Yaskawa INFORM job: DEMO_ROOF_SIDE_0625_3.JBI

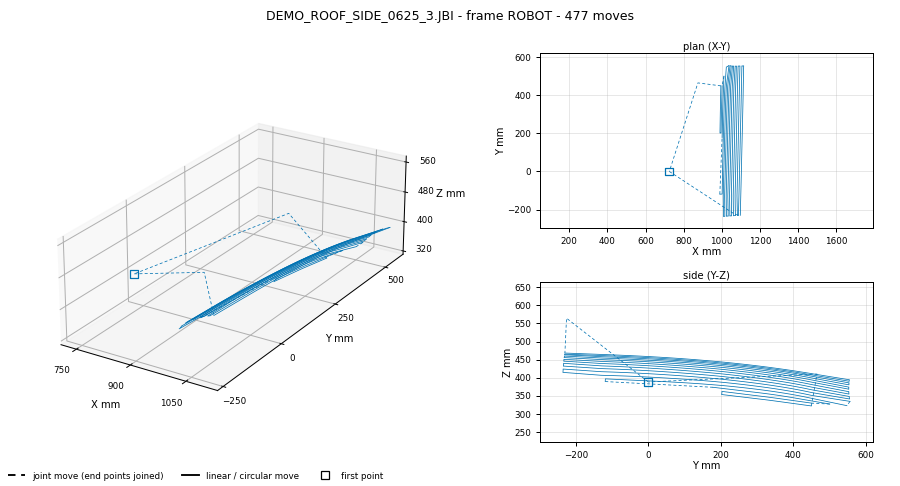
[picture p0: tool path of DEMO_ROOF_SIDE_0625_3.JBI in frame ROBOT, 477 of 477 moves have a stored position in this frame; points joined in program order, loops and branches not executed]
/JOB
//NAME DEMO_ROOF_SIDE_0625_3
//POS
///NPOS 477,0,0,0,0,0
///TOOL 0
///USER 0
///POSTYPE ROBOT
///RECTAN
///RCONF 1,0,0,0,0,0,0,0,0,0,0,0,0,0,0,0,0,0,0,0,0,0,0,0
C00000=725.000,0.000,388.500,-180.000,-0.000,0.000
///USER 0
///POSTYPE ROBOT
///RECTAN
C00001=1070.165,-225.804,564.348,177.658,-15.895,-0.730
C00002=1097.475,-230.239,468.252,177.658,-15.895,-0.730
C00003=1100.518,-106.522,463.583,177.658,-15.895,-0.730
C00004=1101.131,-81.381,462.555,177.457,-15.868,-0.652
C00005=1101.733,-56.230,461.444,177.242,-15.858,-0.568
C00006=1102.322,-31.102,460.246,177.018,-15.859,-0.492
C00007=1102.894,-6.471,458.979,176.786,-15.861,-0.417
C00008=1103.450,17.667,457.639,176.549,-15.857,-0.346
C00009=1103.994,41.321,456.228,176.307,-15.841,-0.282
C00010=1104.527,64.471,454.750,176.060,-15.805,-0.220
C00011=1105.052,87.116,453.204,175.808,-15.748,-0.164
C00012=1105.569,109.258,451.595,175.550,-15.665,-0.106
C00013=1106.076,130.831,449.928,175.291,-15.558,-0.055
C00014=1106.579,151.961,448.197,175.027,-15.428,-0.007
C00015=1107.074,172.585,446.411,174.761,-15.276,0.037
C00016=1107.562,192.652,444.578,174.493,-15.108,0.083
C00017=1107.979,209.697,442.942,174.219,-14.948,0.167
C00018=1108.302,223.398,441.579,174.012,-14.865,0.226
C00019=1108.743,242.055,439.641,173.727,-14.761,0.293
C00020=1109.169,260.166,437.673,173.443,-14.671,0.359
C00021=1109.576,277.536,435.703,173.164,-14.597,0.432
C00022=1109.980,294.921,433.649,172.877,-14.541,0.511
C00023=1110.375,312.126,431.533,172.586,-14.508,0.594
C00024=1110.754,328.858,429.397,172.296,-14.503,0.687
C00025=1111.108,344.779,427.292,172.012,-14.528,0.783
C00026=1111.443,360.182,425.185,171.727,-14.588,0.893
C00027=1111.759,375.112,423.077,171.442,-14.686,1.009
C00028=1112.046,389.128,421.040,171.165,-14.822,1.140
C00029=1112.303,402.245,419.083,170.893,-14.997,1.282
C00030=1112.529,414.390,417.227,170.620,-15.203,1.466
C00031=1112.829,431.883,414.478,170.211,-15.618,1.704
C00032=1112.994,442.551,412.752,169.934,-15.944,1.913
C00033=1113.129,452.452,411.121,169.867,-16.412,1.571
C00034=1115.209,553.765,394.636,169.867,-16.412,1.571
C00035=1105.880,553.291,390.560,169.867,-16.412,1.571
C00036=1103.548,452.102,407.760,170.054,-16.524,0.911
C00037=1103.388,442.223,409.459,170.213,-16.114,0.900
C00038=1103.203,431.578,411.246,170.442,-15.758,0.852
C00039=1103.095,425.743,412.205,170.567,-15.593,0.818
C00040=1102.875,414.111,414.077,170.805,-15.314,0.762
C00041=1102.635,401.997,415.975,171.043,-15.085,0.705
C00042=1102.366,388.898,417.968,171.291,-14.896,0.647
C00043=1102.069,374.899,420.034,171.548,-14.747,0.593
C00044=1101.745,359.987,422.164,171.815,-14.637,0.542
C00045=1101.405,344.600,424.286,172.084,-14.567,0.497
C00046=1101.047,328.694,426.405,172.354,-14.533,0.455
C00047=1100.666,311.978,428.548,172.631,-14.531,0.417
C00048=1100.269,294.786,430.667,172.910,-14.557,0.381
C00049=1099.865,277.416,432.721,173.185,-14.607,0.348
C00050=1099.459,260.059,434.689,173.454,-14.675,0.317
C00051=1099.033,241.963,436.653,173.728,-14.762,0.287
C00052=1098.594,223.318,438.585,174.004,-14.862,0.256
C00053=1098.272,209.617,439.948,174.202,-14.941,0.233
C00054=1097.859,192.596,441.565,174.459,-15.096,0.211
C00055=1097.377,172.542,443.383,174.722,-15.263,0.186
C00056=1096.886,151.931,445.156,174.983,-15.414,0.158
C00057=1096.387,130.814,446.876,175.242,-15.544,0.128
C00058=1095.880,109.241,448.536,175.496,-15.650,0.094
C00059=1095.365,87.114,450.143,175.748,-15.732,0.058
C00060=1094.841,64.483,451.688,175.995,-15.790,0.019
C00061=1094.306,41.347,453.169,176.236,-15.824,-0.022
C00062=1093.761,17.708,454.585,176.472,-15.841,-0.065
C00063=1093.202,-6.416,455.932,176.701,-15.844,-0.107
C00064=1092.628,-31.032,457.209,176.924,-15.841,-0.148
C00065=1092.035,-56.147,458.416,177.138,-15.840,-0.185
C00066=1091.433,-81.271,459.530,177.338,-15.849,-0.214
C00067=1090.821,-106.401,460.556,177.519,-15.875,-0.223
C00068=1087.825,-230.592,465.270,177.627,-15.905,-0.084
C00069=1082.226,-231.045,463.513,177.619,-15.904,-0.053
C00070=1080.117,-128.026,458.207,177.788,-18.751,-0.644
C00071=1080.712,-103.412,457.271,177.590,-18.756,-0.572
C00072=1081.269,-80.191,456.312,177.387,-18.785,-0.479
C00073=1081.838,-56.094,455.234,177.168,-18.840,-0.381
C00074=1082.398,-31.914,454.063,176.940,-18.915,-0.284
C00075=1082.945,-7.981,452.812,176.706,-19.000,-0.187
C00076=1083.496,16.375,451.444,176.461,-19.092,-0.091
C00077=1084.037,40.477,449.991,176.212,-19.178,-0.000
C00078=1084.553,63.576,448.505,175.965,-19.251,0.090
C00079=1085.072,86.781,446.916,175.707,-19.310,0.180
C00080=1085.565,108.870,445.310,175.452,-19.348,0.267
C00081=1086.061,131.068,443.602,175.187,-19.367,0.355
C00082=1086.534,152.148,441.887,174.923,-19.366,0.439
C00083=1087.008,173.221,440.078,174.650,-19.349,0.524
C00084=1087.464,193.399,438.254,174.377,-19.320,0.605
C00085=1087.825,209.395,436.742,174.074,-19.286,0.725
C00086=1088.182,225.416,435.143,173.821,-19.308,0.819
C00087=1088.592,243.865,433.219,173.522,-19.338,0.924
C00088=1089.002,262.278,431.205,173.214,-19.372,1.033
C00089=1089.399,280.152,429.159,172.905,-19.415,1.143
C00090=1089.786,297.588,427.075,172.594,-19.469,1.257
C00091=1090.152,314.076,425.019,172.286,-19.535,1.380
C00092=1090.514,330.569,422.878,171.969,-19.624,1.504
C00093=1090.865,346.565,420.717,171.645,-19.736,1.643
C00094=1091.178,361.013,418.691,171.337,-19.865,1.785
C00095=1091.488,375.512,416.582,171.014,-20.031,1.934
C00096=1091.776,389.121,414.533,170.690,-20.226,2.100
C00097=1092.039,401.783,412.560,170.369,-20.450,2.275
C00098=1092.276,413.455,410.683,170.051,-20.704,2.449
C00099=1092.473,423.358,409.042,169.750,-20.957,2.640
C00100=1092.681,434.084,407.209,169.402,-21.286,2.853
C00101=1092.850,443.075,405.627,169.082,-21.612,3.061
C00102=1093.012,451.962,404.020,169.028,-22.108,2.662
C00103=1095.618,553.013,386.060,169.028,-22.108,2.662
C00104=1085.968,552.705,380.579,169.028,-22.108,2.662
C00105=1082.961,451.807,399.317,168.467,-27.285,2.821
C00106=1082.764,442.923,401.001,168.744,-26.842,2.800
C00107=1082.571,434.067,402.629,169.055,-26.469,2.748
C00108=1082.357,424.236,404.377,169.383,-26.117,2.669
C00109=1082.140,414.335,406.080,169.691,-25.812,2.584
C00110=1081.885,402.576,408.036,170.028,-25.504,2.481
C00111=1081.627,390.820,409.924,170.342,-25.243,2.382
C00112=1081.349,378.124,411.892,170.659,-25.004,2.281
C00113=1081.051,364.541,413.925,170.977,-24.787,2.181
C00114=1080.732,350.019,416.018,171.299,-24.590,2.080
C00115=1080.392,334.507,418.168,171.624,-24.411,1.978
C00116=1080.051,318.965,420.239,171.932,-24.254,1.881
C00117=1079.696,302.745,422.315,172.240,-24.111,1.786
C00118=1079.335,286.239,424.342,172.541,-23.978,1.692
C00119=1078.955,268.767,426.399,172.846,-23.847,1.597
C00120=1078.574,251.297,428.367,173.141,-23.722,1.504
C00121=1078.184,233.235,430.313,173.435,-23.593,1.410
C00122=1077.972,223.469,431.328,173.591,-23.524,1.360
C00123=1077.662,209.105,432.776,173.813,-23.421,1.287
C00124=1077.268,190.976,434.497,174.164,-23.354,1.206
C00125=1076.809,169.900,436.402,174.444,-23.276,1.116
C00126=1076.348,148.818,438.211,174.710,-23.191,1.028
C00127=1075.863,126.605,440.020,174.978,-23.092,0.939
C00128=1075.381,104.512,441.722,175.235,-22.981,0.852
C00129=1074.873,81.414,443.402,175.491,-22.854,0.763
C00130=1074.360,58.187,444.995,175.741,-22.715,0.676
C00131=1073.847,35.079,446.485,175.981,-22.572,0.593
C00132=1073.327,11.848,447.891,176.217,-22.427,0.511
C00133=1072.805,-11.255,449.199,176.446,-22.288,0.435
C00134=1072.275,-34.458,450.423,176.669,-22.160,0.365
C00135=1071.739,-57.560,451.554,176.884,-22.052,0.305
C00136=1071.195,-80.670,452.601,177.089,-21.967,0.257
C00137=1070.662,-102.916,453.529,177.273,-21.914,0.231
C00138=1070.057,-128.042,454.489,177.461,-21.888,0.238
C00139=1071.695,-231.567,459.915,177.355,-21.861,0.543
C00140=1061.501,-232.092,455.769,177.350,-21.861,0.556
C00141=1060.147,-128.074,450.149,177.673,-25.493,-0.352
C00142=1060.424,-116.502,449.716,177.561,-25.496,-0.306
C00143=1060.951,-94.862,448.854,177.335,-25.521,-0.191
C00144=1061.460,-73.669,447.935,177.106,-25.578,-0.067
C00145=1061.974,-51.990,446.914,176.870,-25.664,0.054
C00146=1062.492,-29.881,445.792,176.628,-25.776,0.181
C00147=1063.006,-7.714,444.584,176.382,-25.909,0.311
C00148=1063.527,14.959,443.259,176.128,-26.061,0.445
C00149=1064.053,38.144,441.813,175.866,-26.225,0.588
C00150=1064.574,61.324,440.273,175.600,-26.394,0.727
C00151=1065.091,84.498,438.639,175.330,-26.562,0.869
C00152=1065.593,107.167,436.947,175.056,-26.723,1.016
C00153=1066.079,129.265,435.203,174.777,-26.874,1.165
C00154=1066.552,150.925,433.402,174.490,-27.018,1.316
C00155=1067.011,172.078,431.549,174.196,-27.155,1.468
C00156=1067.457,192.659,429.652,173.895,-27.288,1.615
C00157=1067.805,208.750,428.099,173.466,-27.386,1.843
C00158=1068.310,232.062,425.676,173.073,-27.623,2.036
C00159=1068.730,251.306,423.568,172.729,-27.809,2.207
C00160=1069.116,268.867,421.555,172.398,-27.974,2.377
C00161=1069.505,286.433,419.452,172.047,-28.138,2.558
C00162=1069.874,303.035,417.377,171.699,-28.297,2.739
C00163=1070.242,319.454,415.238,171.336,-28.464,2.927
C00164=1070.595,335.095,413.114,170.965,-28.634,3.123
C00165=1070.927,349.716,411.048,170.598,-28.812,3.311
C00166=1071.240,363.349,409.047,170.224,-28.996,3.517
C00167=1071.559,377.040,406.959,169.821,-29.207,3.734
C00168=1071.859,389.849,404.929,169.410,-29.434,3.960
C00169=1072.142,401.720,402.976,168.993,-29.677,4.190
C00170=1072.406,412.613,401.117,168.564,-29.930,4.439
C00171=1072.674,423.498,399.190,168.090,-30.222,4.706
C00172=1072.925,433.455,397.359,167.603,-30.529,4.984
C00173=1073.167,442.803,395.573,167.144,-30.880,5.170
C00174=1073.417,451.686,393.819,167.000,-31.383,4.760
C00175=1076.941,552.431,374.355,167.000,-31.383,4.760
C00176=1070.604,552.364,368.674,167.000,-31.383,4.760
C00177=1064.303,450.677,387.868,166.732,-35.182,4.427
C00178=1063.991,441.090,389.826,167.182,-34.765,4.439
C00179=1063.720,432.199,391.572,167.581,-34.434,4.400
C00180=1063.453,423.074,393.298,167.968,-34.139,4.326
C00181=1063.171,413.034,395.127,168.363,-33.856,4.229
C00182=1062.875,402.145,397.038,168.761,-33.591,4.109
C00183=1062.585,391.123,398.901,169.134,-33.357,3.985
C00184=1062.277,379.170,400.848,169.505,-33.134,3.857
C00185=1061.955,366.340,402.861,169.871,-32.924,3.727
C00186=1061.623,352.844,404.897,170.232,-32.729,3.590
C00187=1061.284,338.827,406.933,170.580,-32.548,3.454
C00188=1060.933,324.057,408.996,170.921,-32.374,3.318
C00189=1060.562,308.264,411.115,171.264,-32.203,3.179
C00190=1060.195,292.480,413.150,171.585,-32.039,3.045
C00191=1059.791,274.985,415.313,171.923,-31.862,2.901
C00192=1059.578,265.654,416.429,172.096,-31.768,2.826
C00193=1059.153,246.982,418.589,172.428,-31.577,2.677
C00194=1058.723,227.872,420.701,172.753,-31.373,2.528
C00195=1058.283,208.328,422.764,173.071,-31.153,2.375
C00196=1057.996,195.285,424.047,173.443,-31.051,2.282
C00197=1057.574,176.199,425.849,173.723,-30.911,2.154
C00198=1057.126,155.969,427.670,174.001,-30.768,2.025
C00199=1056.654,134.875,429.477,174.275,-30.621,1.897
C00200=1056.157,112.776,431.275,174.547,-30.468,1.768
C00201=1055.652,90.530,432.991,174.809,-30.313,1.642
C00202=1055.123,67.421,434.676,175.073,-30.153,1.517
C00203=1054.608,45.164,436.208,175.322,-30.002,1.402
C00204=1054.092,23.041,437.644,175.565,-29.858,1.293
C00205=1053.572,0.919,438.994,175.807,-29.724,1.189
C00206=1053.043,-21.324,440.263,176.047,-29.606,1.091
C00207=1052.537,-42.438,441.385,176.272,-29.511,1.008
C00208=1052.052,-62.559,442.379,176.482,-29.443,0.939
C00209=1051.536,-83.822,443.351,176.696,-29.396,0.884
C00210=1051.017,-104.972,444.237,176.893,-29.379,0.856
C00211=1050.452,-128.121,445.120,177.078,-29.394,0.882
C00212=1051.564,-232.631,450.944,176.858,-29.343,1.365
C00213=1042.728,-233.148,445.881,176.855,-29.343,1.373
C00214=1041.055,-129.188,439.415,176.733,-33.542,1.452
C00215=1041.065,-127.686,439.343,177.520,-33.611,0.006
C00216=1041.589,-106.531,438.551,177.251,-33.551,0.150
C00217=1042.089,-86.375,437.718,176.986,-33.524,0.299
C00218=1042.591,-66.101,436.801,176.722,-33.523,0.444
C00219=1043.089,-45.974,435.813,176.456,-33.546,0.600
C00220=1043.609,-24.854,434.695,176.181,-33.593,0.760
C00221=1044.128,-3.735,433.493,175.906,-33.658,0.928
C00222=1044.670,18.526,432.137,175.625,-33.744,1.095
C00223=1045.207,40.652,430.701,175.342,-33.840,1.273
C00224=1045.742,62.918,429.165,175.060,-33.945,1.448
C00225=1046.270,85.031,427.551,174.774,-34.054,1.631
C00226=1046.792,107.138,425.848,174.479,-34.165,1.821
C00227=1047.313,129.384,424.039,174.171,-34.278,2.020
C00228=1047.801,150.481,422.232,173.868,-34.388,2.208
C00229=1048.265,170.574,420.425,173.553,-34.495,2.410
C00230=1048.725,190.660,418.527,173.225,-34.608,2.606
C00231=1049.118,207.841,416.825,172.677,-34.707,2.857
C00232=1049.329,216.744,415.881,172.491,-34.790,3.008
C00233=1049.776,235.626,413.812,172.148,-34.968,3.221
C00234=1050.223,254.375,411.667,171.786,-35.132,3.443
C00235=1050.650,272.185,409.542,171.416,-35.279,3.673
C00236=1051.080,290.001,407.322,171.023,-35.423,3.908
C00237=1051.493,306.884,405.125,170.626,-35.562,4.139
C00238=1051.889,322.821,402.963,170.218,-35.698,4.379
C00239=1052.266,337.737,400.856,169.805,-35.833,4.618
C00240=1052.624,351.637,398.812,169.387,-35.971,4.855
C00241=1052.992,365.548,396.685,168.951,-36.131,5.079
C00242=1053.165,372.035,395.661,168.703,-36.204,5.241
C00243=1053.512,384.546,393.629,168.231,-36.370,5.500
C00244=1053.841,396.047,391.687,167.744,-36.540,5.774
C00245=1054.169,407.125,389.742,167.264,-36.737,5.999
C00246=1054.341,412.713,388.730,166.953,-36.832,6.202
C00247=1054.666,422.922,386.827,166.395,-37.039,6.496
C00248=1054.977,432.221,385.023,165.818,-37.249,6.805
C00249=1055.291,441.109,383.228,165.236,-37.483,7.070
C00250=1055.624,449.834,381.397,166.221,-38.279,4.713
C00251=1062.727,552.413,361.747,166.099,-38.338,4.732
C00252=1056.155,552.786,355.236,166.099,-38.338,4.732
C00253=1047.397,450.217,374.283,165.269,-40.798,5.659
C00254=1047.334,449.231,374.484,165.320,-40.769,5.670
C00255=1046.948,440.387,376.373,165.757,-40.480,5.763
C00256=1046.608,431.889,378.121,166.167,-40.241,5.783
C00257=1046.237,422.009,380.072,166.634,-40.007,5.732
C00258=1045.869,411.615,382.039,167.096,-39.798,5.641
C00259=1045.521,401.242,383.924,167.530,-39.619,5.523
C00260=1045.161,389.952,385.897,167.965,-39.451,5.385
C00261=1044.798,378.069,387.892,168.385,-39.298,5.244
C00262=1044.412,364.913,390.012,168.808,-39.152,5.094
C00263=1044.041,351.826,392.037,169.199,-39.027,4.938
C00264=1043.655,337.762,394.130,169.584,-38.909,4.780
C00265=1043.251,322.681,396.284,169.963,-38.797,4.618
C00266=1042.854,307.576,398.355,170.315,-38.697,4.462
C00267=1042.436,291.367,400.490,170.665,-38.596,4.300
C00268=1042.003,274.390,402.637,171.006,-38.495,4.136
C00269=1041.548,256.427,404.814,171.344,-38.389,3.966
C00270=1041.070,237.456,407.017,171.680,-38.273,3.789
C00271=1040.591,218.337,409.144,172.000,-38.147,3.612
C00272=1040.313,207.289,410.334,172.178,-38.069,3.509
C00273=1039.855,188.107,412.240,172.741,-38.010,3.347
C00274=1039.375,168.021,414.138,173.049,-37.960,3.188
C00275=1038.893,147.927,415.944,173.335,-37.919,3.039
C00276=1038.383,126.831,417.748,173.615,-37.881,2.889
C00277=1037.841,104.582,419.554,173.896,-37.845,2.738
C00278=1037.297,82.475,421.254,174.165,-37.815,2.593
C00279=1036.743,60.213,422.873,174.429,-37.788,2.453
C00280=1036.190,38.092,424.392,174.688,-37.767,2.319
C00281=1035.632,15.964,425.821,174.947,-37.757,2.190
C00282=1035.094,-5.300,427.107,175.197,-37.758,2.072
C00283=1034.559,-26.422,428.301,175.445,-37.774,1.964
C00284=1034.023,-47.545,429.407,175.693,-37.808,1.866
C00285=1033.509,-67.808,430.385,175.925,-37.861,1.787
C00286=1033.028,-86.955,431.234,176.133,-37.930,1.735
C00287=1032.523,-107.114,432.049,176.328,-38.025,1.718
C00288=1032.000,-128.274,432.819,176.486,-38.148,1.775
C00289=1032.002,-130.279,432.929,176.497,-38.132,1.787
C00290=1033.937,-233.693,439.953,176.074,-38.077,2.488
C00291=1024.589,-234.330,432.344,176.066,-38.077,2.501
C00292=1023.346,-129.891,425.429,176.234,-43.473,2.146
C00293=1023.362,-127.890,425.334,177.376,-43.542,0.462
C00294=1023.884,-106.728,424.604,177.047,-43.318,0.656
C00295=1024.389,-86.569,423.824,176.729,-43.122,0.846
C00296=1024.878,-67.290,422.998,176.426,-42.953,1.029
C00297=1025.394,-47.161,422.055,176.107,-42.791,1.231
C00298=1025.940,-26.038,420.976,175.787,-42.637,1.430
C00299=1026.488,-4.917,419.808,175.474,-42.497,1.630
C00300=1027.041,16.348,418.545,175.163,-42.367,1.835
C00301=1027.615,38.474,417.138,174.851,-42.242,2.042
C00302=1028.188,60.594,415.640,174.538,-42.123,2.257
C00303=1028.759,82.853,414.040,174.229,-42.011,2.466
C00304=1029.322,104.959,412.359,173.909,-41.902,2.690
C00305=1029.885,127.205,410.570,173.577,-41.796,2.918
C00306=1030.412,148.301,408.779,173.247,-41.701,3.141
C00307=1030.925,168.908,406.937,172.904,-41.615,3.369
C00308=1031.411,188.478,405.096,172.545,-41.540,3.606
C00309=1031.863,206.668,403.296,171.800,-41.466,3.995
C00310=1032.406,227.136,401.068,171.427,-41.483,4.257
C00311=1032.913,246.305,398.887,171.058,-41.495,4.503
C00312=1033.401,264.682,396.707,170.669,-41.503,4.761
C00313=1033.859,281.837,394.582,170.277,-41.512,5.014
C00314=1034.295,298.037,392.492,169.874,-41.523,5.271
C00315=1034.740,314.296,390.304,169.438,-41.541,5.539
C00316=1035.166,329.577,388.161,168.991,-41.567,5.807
C00317=1035.575,343.840,386.075,168.537,-41.601,6.071
C00318=1035.966,357.090,384.058,168.073,-41.643,6.337
C00319=1036.342,369.364,382.115,167.602,-41.692,6.601
C00320=1036.736,381.713,380.082,167.080,-41.753,6.888
C00321=1037.120,393.199,378.112,166.545,-41.824,7.174
C00322=1037.502,404.081,376.169,165.981,-41.902,7.470
C00323=1037.896,414.646,374.203,165.379,-41.993,7.775
C00324=1038.276,424.250,372.342,164.772,-42.087,8.072
C00325=1038.650,433.139,370.549,164.136,-42.181,8.385
C00326=1039.050,442.014,368.684,163.581,-42.332,8.497
C00327=1039.386,448.734,367.229,164.760,-42.968,6.160
C00328=1039.554,450.903,366.800,166.209,-43.445,3.844
C00329=1049.939,553.476,348.598,166.075,-43.471,3.853
C00330=1043.749,554.518,341.634,166.075,-43.471,3.853
C00331=1031.999,451.287,359.121,164.131,-44.920,6.554
C00332=1031.817,449.308,359.493,164.232,-44.897,6.597
C00333=1031.673,447.334,359.896,164.324,-44.866,6.647
C00334=1031.258,439.448,361.609,164.670,-44.716,6.833
C00335=1030.831,430.598,363.461,165.080,-44.583,6.928
C00336=1030.393,420.786,365.428,165.551,-44.475,6.922
C00337=1029.980,410.902,367.328,166.013,-44.394,6.857
C00338=1029.558,400.128,369.312,166.484,-44.327,6.759
C00339=1029.158,389.280,371.231,166.924,-44.279,6.647
C00340=1028.759,377.884,373.165,167.351,-44.248,6.521
C00341=1028.363,365.992,375.105,167.761,-44.231,6.388
C00342=1027.966,353.521,377.060,168.157,-44.229,6.250
C00343=1027.552,340.075,379.084,168.549,-44.243,6.103
C00344=1027.153,326.610,381.031,168.909,-44.271,5.962
C00345=1026.734,312.130,383.043,169.263,-44.316,5.815
C00346=1026.295,296.672,385.103,169.612,-44.378,5.667
C00347=1025.838,280.282,387.198,169.949,-44.457,5.516
C00348=1025.374,263.513,389.252,170.267,-44.550,5.367
C00349=1024.897,246.176,391.288,170.573,-44.658,5.216
C00350=1024.393,227.814,393.355,170.873,-44.784,5.060
C00351=1023.789,205.974,395.701,171.208,-44.948,4.873
C00352=1023.326,187.781,397.459,171.828,-45.167,4.730
C00353=1022.841,168.692,399.210,172.114,-45.408,4.595
C00354=1022.347,149.197,400.908,172.379,-45.664,4.467
C00355=1021.821,128.504,402.618,172.639,-45.938,4.337
C00356=1021.252,106.263,404.357,172.900,-46.238,4.205
C00357=1020.681,84.159,405.987,173.148,-46.539,4.078
C00358=1020.106,62.049,407.524,173.392,-46.842,3.953
C00359=1019.525,39.788,408.977,173.637,-47.150,3.830
C00360=1018.972,18.663,410.270,173.871,-47.445,3.714
C00361=1018.420,-2.461,411.478,174.109,-47.744,3.602
C00362=1017.868,-23.710,412.603,174.350,-48.051,3.497
C00363=1017.323,-44.829,413.632,174.588,-48.362,3.405
C00364=1016.811,-64.954,414.526,174.811,-48.668,3.331
C00365=1016.306,-85.225,415.343,175.018,-48.982,3.284
C00366=1015.812,-105.379,416.068,175.191,-49.301,3.282
C00367=1015.262,-128.538,416.803,175.315,-49.671,3.378
C00368=1015.251,-130.539,416.903,175.316,-49.672,3.399
C00369=1016.357,-234.959,424.092,174.502,-49.579,4.489
C00370=1009.142,-235.587,414.945,174.483,-49.577,4.514
C00371=1007.924,-132.221,407.110,173.437,-57.121,5.689
C00372=1007.919,-130.220,406.985,175.670,-57.272,3.016
C00373=1007.941,-128.219,406.903,177.234,-57.313,1.139
C00374=1008.429,-106.073,406.307,176.821,-56.772,1.422
C00375=1008.916,-84.803,405.643,176.411,-56.240,1.708
C00376=1009.413,-63.677,404.890,176.025,-55.709,1.971
C00377=1009.923,-42.559,404.047,175.648,-55.173,2.230
C00378=1010.440,-21.563,403.120,175.285,-54.640,2.482
C00379=1010.973,-0.216,402.086,174.929,-54.099,2.733
C00380=1011.528,21.902,400.920,174.588,-53.536,2.969
C00381=1012.090,44.157,399.654,174.267,-52.965,3.190
C00382=1012.650,66.270,398.304,173.947,-52.390,3.413
C00383=1013.207,88.376,396.862,173.631,-51.812,3.633
C00384=1013.740,109.616,395.385,173.330,-51.254,3.837
C00385=1014.242,129.717,393.903,173.025,-50.724,4.046
C00386=1014.742,149.813,392.336,172.707,-50.196,4.255
C00387=1015.216,168.908,390.761,172.380,-49.697,4.467
C00388=1015.692,187.997,389.098,172.032,-49.205,4.681
C00389=1016.124,205.183,387.516,171.128,-48.746,5.162
C00390=1016.691,225.453,385.421,170.756,-48.339,5.405
C00391=1017.151,242.031,383.624,170.418,-48.032,5.630
C00392=1017.612,258.578,381.752,170.050,-47.747,5.874
C00393=1018.044,274.118,379.916,169.679,-47.498,6.113
C00394=1018.482,289.671,377.999,169.282,-47.269,6.362
C00395=1018.899,304.273,376.122,168.878,-47.070,6.608
C00396=1019.327,318.937,374.156,168.438,-46.886,6.871
C00397=1019.737,332.627,372.241,167.990,-46.729,7.135
C00398=1020.161,346.293,370.248,167.513,-46.589,7.399
C00399=1020.569,358.948,368.324,167.018,-46.469,7.678
C00400=1020.996,371.625,366.312,166.491,-46.365,7.951
C00401=1021.415,383.389,364.365,165.941,-46.275,8.241
C00402=1021.823,394.279,362.486,165.388,-46.203,8.516
C00403=1022.258,405.184,360.525,164.778,-46.138,8.815
C00404=1022.709,415.757,358.539,164.132,-46.083,9.111
C00405=1023.135,425.067,356.715,163.493,-46.037,9.403
C00406=1023.579,434.107,354.868,162.815,-45.995,9.697
C00407=1024.053,443.067,352.959,162.434,-46.065,9.500
C00408=1024.290,447.008,352.107,163.950,-46.590,7.057
C00409=1024.540,449.974,351.528,165.626,-47.071,4.488
C00410=1024.865,452.950,351.010,167.064,-47.437,2.246
C00411=1038.281,555.950,334.991,166.893,-47.426,2.243
C00412=1024.102,547.273,323.190,166.893,-47.426,2.243
C00413=1016.966,444.029,344.663,163.713,-48.167,7.630
C00414=1016.501,435.747,346.429,164.086,-48.176,7.802
C00415=1016.019,426.476,348.324,164.512,-48.211,7.900
C00416=1015.545,416.591,350.257,164.960,-48.270,7.932
C00417=1015.089,406.366,352.169,165.395,-48.349,7.931
C00418=1014.668,396.230,353.986,165.798,-48.442,7.907
C00419=1014.243,385.335,355.859,166.214,-48.561,7.849
C00420=1013.805,373.353,357.831,166.642,-48.711,7.765
C00421=1013.393,361.454,359.704,167.036,-48.877,7.674
C00422=1013.002,349.576,361.497,167.398,-49.061,7.583
C00423=1012.597,336.690,363.362,167.758,-49.280,7.486
C00424=1012.236,324.767,365.017,168.063,-49.500,7.402
C00425=1011.857,311.853,366.740,168.365,-49.759,7.318
C00426=1011.461,297.964,368.514,168.660,-50.060,7.238
C00427=1011.074,284.057,370.214,168.922,-50.388,7.173
C00428=1010.698,270.357,371.820,169.146,-50.735,7.131
C00429=1010.299,255.595,373.474,169.369,-51.141,7.087
C00430=1009.902,240.819,375.057,169.576,-51.583,7.045
C00431=1009.506,226.014,376.573,169.763,-52.061,7.010
C00432=1009.135,212.167,377.926,169.920,-52.545,6.987
C00433=1008.923,204.277,378.672,170.007,-52.837,6.972
C00434=1008.783,198.223,379.190,170.459,-53.095,6.974
C00435=1008.447,183.688,380.390,170.598,-53.719,6.977
C00436=1008.047,166.092,381.767,170.734,-54.479,6.991
C00437=1007.629,147.559,383.133,170.848,-55.283,7.015
C00438=1007.199,128.396,384.461,170.941,-56.116,7.047
C00439=1006.746,108.166,385.778,171.018,-56.988,7.087
C00440=1006.263,86.565,387.094,171.083,-57.906,7.134
C00441=1006.016,75.514,387.733,171.107,-58.365,7.167
C00442=1005.500,52.287,389.002,171.172,-59.303,7.209
C00443=1004.990,29.177,390.172,171.244,-60.180,7.239
C00444=1004.487,5.948,391.259,171.337,-60.982,7.247
C00445=1004.019,-16.153,392.215,171.450,-61.648,7.230
C00446=1002.098,-118.686,397.119,172.117,-61.700,6.473
C00447=990.034,-119.072,389.643,172.117,-61.700,6.473
C00448=1001.913,178.181,373.829,169.046,-61.424,9.964
C00449=1004.146,280.106,361.704,169.054,-53.702,7.479
C00450=1004.435,291.519,360.402,168.703,-53.278,7.685
C00451=1004.778,304.570,358.847,168.295,-52.818,7.915
C00452=1005.135,317.689,357.209,167.868,-52.379,8.143
C00453=1005.507,330.827,355.491,167.413,-51.962,8.381
C00454=1005.867,342.948,353.830,166.967,-51.596,8.606
C00455=1006.245,355.054,352.097,166.487,-51.248,8.844
C00456=1006.605,365.978,350.464,166.020,-50.946,9.070
C00457=1006.994,377.108,348.729,165.509,-50.650,9.310
C00458=1007.402,388.096,346.941,164.946,-50.364,9.579
C00459=1007.836,398.997,345.084,164.398,-50.103,9.782
C00460=1011.634,500.093,327.595,164.398,-50.103,9.782
C00461=1001.995,450.158,330.138,164.398,-50.103,9.782
C00462=999.492,348.504,344.304,166.915,-52.970,8.838
C00463=999.147,335.929,346.007,167.247,-53.328,8.804
C00464=998.829,323.558,347.604,167.551,-53.695,8.768
C00465=998.516,310.614,349.197,167.843,-54.091,8.733
C00466=998.385,304.901,349.876,167.958,-54.269,8.726
C00467=996.342,203.024,362.425,168.899,-54.407,7.568
C00468=990.898,202.057,353.878,168.878,-54.404,7.594
C00469=992.419,303.989,341.703,168.394,-54.335,8.189
C00470=992.522,309.706,341.045,168.112,-54.133,8.401
C00471=992.777,322.617,339.499,167.649,-53.711,8.646
C00472=993.043,334.958,337.943,167.180,-53.317,8.888
C00473=993.338,347.503,336.283,166.622,-52.918,9.206
C00474=995.437,449.208,322.419,166.622,-52.918,9.206
C00475=874.966,464.843,410.409,166.622,-52.918,9.206
///USER 0
///POSTYPE ROBOT
///RECTAN
C00476=725.000,0.000,388.500,-180.000,-0.000,0.000
//INST
///DATE 2021/06/25 12:02
///ATTR SC,RW,RJ
////FRAME ROBOT
///GROUP1 RB1
NOP
MOVJ C00000 VJ=25.00 PL=0
'Path Start: side
MOVJ C00001 VJ=25.00 PL=0
MOVJ C00002 VJ=25.00 PL=0
SPYON
MOVL C00003 V=800.0 PL=8
MOVL C00004 V=800.0 PL=8
MOVL C00005 V=800.0 PL=8
MOVL C00006 V=800.0 PL=8
MOVL C00007 V=800.0 PL=8
MOVL C00008 V=800.0 PL=8
MOVL C00009 V=800.0 PL=8
MOVL C00010 V=800.0 PL=8
MOVL C00011 V=800.0 PL=8
MOVL C00012 V=800.0 PL=8
MOVL C00013 V=800.0 PL=8
MOVL C00014 V=800.0 PL=8
MOVL C00015 V=800.0 PL=8
MOVL C00016 V=800.0 PL=8
MOVL C00017 V=800.0 PL=8
MOVL C00018 V=800.0 PL=8
MOVL C00019 V=800.0 PL=8
MOVL C00020 V=800.0 PL=8
MOVL C00021 V=800.0 PL=8
MOVL C00022 V=800.0 PL=8
MOVL C00023 V=800.0 PL=8
MOVL C00024 V=800.0 PL=8
MOVL C00025 V=800.0 PL=8
MOVL C00026 V=800.0 PL=8
MOVL C00027 V=800.0 PL=8
MOVL C00028 V=800.0 PL=8
MOVL C00029 V=800.0 PL=8
MOVL C00030 V=800.0 PL=8
MOVL C00031 V=800.0 PL=8
MOVL C00032 V=800.0 PL=8
MOVL C00033 V=800.0 PL=8
MOVL C00034 V=800.0 PL=0
SPYOF
MOVJ C00035 VJ=25.00 PL=0
SPYON
MOVL C00036 V=800.0 PL=8
MOVL C00037 V=800.0 PL=8
MOVL C00038 V=800.0 PL=8
MOVL C00039 V=800.0 PL=8
MOVL C00040 V=800.0 PL=8
MOVL C00041 V=800.0 PL=8
MOVL C00042 V=800.0 PL=8
MOVL C00043 V=800.0 PL=8
MOVL C00044 V=800.0 PL=8
MOVL C00045 V=800.0 PL=8
MOVL C00046 V=800.0 PL=8
MOVL C00047 V=800.0 PL=8
MOVL C00048 V=800.0 PL=8
MOVL C00049 V=800.0 PL=8
MOVL C00050 V=800.0 PL=8
MOVL C00051 V=800.0 PL=8
MOVL C00052 V=800.0 PL=8
MOVL C00053 V=800.0 PL=8
MOVL C00054 V=800.0 PL=8
MOVL C00055 V=800.0 PL=8
MOVL C00056 V=800.0 PL=8
MOVL C00057 V=800.0 PL=8
MOVL C00058 V=800.0 PL=8
MOVL C00059 V=800.0 PL=8
MOVL C00060 V=800.0 PL=8
MOVL C00061 V=800.0 PL=8
MOVL C00062 V=800.0 PL=8
MOVL C00063 V=800.0 PL=8
MOVL C00064 V=800.0 PL=8
MOVL C00065 V=800.0 PL=8
MOVL C00066 V=800.0 PL=8
MOVL C00067 V=800.0 PL=8
MOVL C00068 V=800.0 PL=0
SPYOF
MOVJ C00069 VJ=25.00 PL=0
SPYON
MOVL C00070 V=800.0 PL=8
MOVL C00071 V=800.0 PL=8
MOVL C00072 V=800.0 PL=8
MOVL C00073 V=800.0 PL=8
MOVL C00074 V=800.0 PL=8
MOVL C00075 V=800.0 PL=8
MOVL C00076 V=800.0 PL=8
MOVL C00077 V=800.0 PL=8
MOVL C00078 V=800.0 PL=8
MOVL C00079 V=800.0 PL=8
MOVL C00080 V=800.0 PL=8
MOVL C00081 V=800.0 PL=8
MOVL C00082 V=800.0 PL=8
MOVL C00083 V=800.0 PL=8
MOVL C00084 V=800.0 PL=8
MOVL C00085 V=800.0 PL=8
MOVL C00086 V=800.0 PL=8
MOVL C00087 V=800.0 PL=8
MOVL C00088 V=800.0 PL=8
MOVL C00089 V=800.0 PL=8
MOVL C00090 V=800.0 PL=8
MOVL C00091 V=800.0 PL=8
MOVL C00092 V=800.0 PL=8
MOVL C00093 V=800.0 PL=8
MOVL C00094 V=800.0 PL=8
MOVL C00095 V=800.0 PL=8
MOVL C00096 V=800.0 PL=8
MOVL C00097 V=800.0 PL=8
MOVL C00098 V=800.0 PL=8
MOVL C00099 V=800.0 PL=8
MOVL C00100 V=800.0 PL=8
MOVL C00101 V=800.0 PL=8
MOVL C00102 V=800.0 PL=8
MOVL C00103 V=800.0 PL=0
SPYOF
MOVJ C00104 VJ=25.00 PL=0
SPYON
MOVL C00105 V=800.0 PL=8
MOVL C00106 V=800.0 PL=8
MOVL C00107 V=800.0 PL=8
MOVL C00108 V=800.0 PL=8
MOVL C00109 V=800.0 PL=8
MOVL C00110 V=800.0 PL=8
MOVL C00111 V=800.0 PL=8
MOVL C00112 V=800.0 PL=8
MOVL C00113 V=800.0 PL=8
MOVL C00114 V=800.0 PL=8
MOVL C00115 V=800.0 PL=8
MOVL C00116 V=800.0 PL=8
MOVL C00117 V=800.0 PL=8
MOVL C00118 V=800.0 PL=8
MOVL C00119 V=800.0 PL=8
MOVL C00120 V=800.0 PL=8
MOVL C00121 V=800.0 PL=8
MOVL C00122 V=800.0 PL=8
MOVL C00123 V=800.0 PL=8
MOVL C00124 V=800.0 PL=8
MOVL C00125 V=800.0 PL=8
MOVL C00126 V=800.0 PL=8
MOVL C00127 V=800.0 PL=8
MOVL C00128 V=800.0 PL=8
MOVL C00129 V=800.0 PL=8
MOVL C00130 V=800.0 PL=8
MOVL C00131 V=800.0 PL=8
MOVL C00132 V=800.0 PL=8
MOVL C00133 V=800.0 PL=8
MOVL C00134 V=800.0 PL=8
MOVL C00135 V=800.0 PL=8
MOVL C00136 V=800.0 PL=8
MOVL C00137 V=800.0 PL=8
MOVL C00138 V=800.0 PL=8
MOVL C00139 V=800.0 PL=0
SPYOF
MOVJ C00140 VJ=25.00 PL=0
SPYON
MOVL C00141 V=800.0 PL=8
MOVL C00142 V=800.0 PL=8
MOVL C00143 V=800.0 PL=8
MOVL C00144 V=800.0 PL=8
MOVL C00145 V=800.0 PL=8
MOVL C00146 V=800.0 PL=8
MOVL C00147 V=800.0 PL=8
MOVL C00148 V=800.0 PL=8
MOVL C00149 V=800.0 PL=8
MOVL C00150 V=800.0 PL=8
MOVL C00151 V=800.0 PL=8
MOVL C00152 V=800.0 PL=8
MOVL C00153 V=800.0 PL=8
MOVL C00154 V=800.0 PL=8
MOVL C00155 V=800.0 PL=8
MOVL C00156 V=800.0 PL=8
MOVL C00157 V=800.0 PL=8
MOVL C00158 V=800.0 PL=8
MOVL C00159 V=800.0 PL=8
MOVL C00160 V=800.0 PL=8
MOVL C00161 V=800.0 PL=8
MOVL C00162 V=800.0 PL=8
MOVL C00163 V=800.0 PL=8
MOVL C00164 V=800.0 PL=8
MOVL C00165 V=800.0 PL=8
MOVL C00166 V=800.0 PL=8
MOVL C00167 V=800.0 PL=8
MOVL C00168 V=800.0 PL=8
MOVL C00169 V=800.0 PL=8
MOVL C00170 V=800.0 PL=8
MOVL C00171 V=800.0 PL=8
MOVL C00172 V=800.0 PL=8
MOVL C00173 V=800.0 PL=8
MOVL C00174 V=800.0 PL=8
MOVL C00175 V=800.0 PL=0
SPYOF
MOVJ C00176 VJ=25.00 PL=0
SPYON
MOVL C00177 V=800.0 PL=8
MOVL C00178 V=800.0 PL=8
MOVL C00179 V=800.0 PL=8
MOVL C00180 V=800.0 PL=8
MOVL C00181 V=800.0 PL=8
MOVL C00182 V=800.0 PL=8
MOVL C00183 V=800.0 PL=8
MOVL C00184 V=800.0 PL=8
MOVL C00185 V=800.0 PL=8
MOVL C00186 V=800.0 PL=8
MOVL C00187 V=800.0 PL=8
MOVL C00188 V=800.0 PL=8
MOVL C00189 V=800.0 PL=8
MOVL C00190 V=800.0 PL=8
MOVL C00191 V=800.0 PL=8
MOVL C00192 V=800.0 PL=8
MOVL C00193 V=800.0 PL=8
MOVL C00194 V=800.0 PL=8
MOVL C00195 V=800.0 PL=8
MOVL C00196 V=800.0 PL=8
MOVL C00197 V=800.0 PL=8
MOVL C00198 V=800.0 PL=8
MOVL C00199 V=800.0 PL=8
MOVL C00200 V=800.0 PL=8
MOVL C00201 V=800.0 PL=8
MOVL C00202 V=800.0 PL=8
MOVL C00203 V=800.0 PL=8
MOVL C00204 V=800.0 PL=8
MOVL C00205 V=800.0 PL=8
MOVL C00206 V=800.0 PL=8
MOVL C00207 V=800.0 PL=8
MOVL C00208 V=800.0 PL=8
MOVL C00209 V=800.0 PL=8
MOVL C00210 V=800.0 PL=8
MOVL C00211 V=800.0 PL=8
MOVL C00212 V=800.0 PL=0
SPYOF
MOVJ C00213 VJ=25.00 PL=0
SPYON
MOVL C00214 V=800.0 PL=8
MOVL C00215 V=800.0 PL=8
MOVL C00216 V=800.0 PL=8
MOVL C00217 V=800.0 PL=8
MOVL C00218 V=800.0 PL=8
MOVL C00219 V=800.0 PL=8
MOVL C00220 V=800.0 PL=8
MOVL C00221 V=800.0 PL=8
MOVL C00222 V=800.0 PL=8
MOVL C00223 V=800.0 PL=8
MOVL C00224 V=800.0 PL=8
MOVL C00225 V=800.0 PL=8
MOVL C00226 V=800.0 PL=8
MOVL C00227 V=800.0 PL=8
MOVL C00228 V=800.0 PL=8
MOVL C00229 V=800.0 PL=8
MOVL C00230 V=800.0 PL=8
MOVL C00231 V=800.0 PL=8
MOVL C00232 V=800.0 PL=8
MOVL C00233 V=800.0 PL=8
MOVL C00234 V=800.0 PL=8
MOVL C00235 V=800.0 PL=8
MOVL C00236 V=800.0 PL=8
MOVL C00237 V=800.0 PL=8
MOVL C00238 V=800.0 PL=8
MOVL C00239 V=800.0 PL=8
MOVL C00240 V=800.0 PL=8
MOVL C00241 V=800.0 PL=8
MOVL C00242 V=800.0 PL=8
MOVL C00243 V=800.0 PL=8
MOVL C00244 V=800.0 PL=8
MOVL C00245 V=800.0 PL=8
MOVL C00246 V=800.0 PL=8
MOVL C00247 V=800.0 PL=8
MOVL C00248 V=800.0 PL=8
MOVL C00249 V=800.0 PL=8
MOVL C00250 V=800.0 PL=8
MOVL C00251 V=800.0 PL=0
SPYOF
MOVJ C00252 VJ=25.00 PL=0
SPYON
MOVL C00253 V=800.0 PL=8
MOVL C00254 V=800.0 PL=8
MOVL C00255 V=800.0 PL=8
MOVL C00256 V=800.0 PL=8
MOVL C00257 V=800.0 PL=8
MOVL C00258 V=800.0 PL=8
MOVL C00259 V=800.0 PL=8
MOVL C00260 V=800.0 PL=8
MOVL C00261 V=800.0 PL=8
MOVL C00262 V=800.0 PL=8
MOVL C00263 V=800.0 PL=8
MOVL C00264 V=800.0 PL=8
MOVL C00265 V=800.0 PL=8
MOVL C00266 V=800.0 PL=8
MOVL C00267 V=800.0 PL=8
MOVL C00268 V=800.0 PL=8
MOVL C00269 V=800.0 PL=8
MOVL C00270 V=800.0 PL=8
MOVL C00271 V=800.0 PL=8
MOVL C00272 V=800.0 PL=8
MOVL C00273 V=800.0 PL=8
MOVL C00274 V=800.0 PL=8
MOVL C00275 V=800.0 PL=8
MOVL C00276 V=800.0 PL=8
MOVL C00277 V=800.0 PL=8
MOVL C00278 V=800.0 PL=8
MOVL C00279 V=800.0 PL=8
MOVL C00280 V=800.0 PL=8
MOVL C00281 V=800.0 PL=8
MOVL C00282 V=800.0 PL=8
MOVL C00283 V=800.0 PL=8
MOVL C00284 V=800.0 PL=8
MOVL C00285 V=800.0 PL=8
MOVL C00286 V=800.0 PL=8
MOVL C00287 V=800.0 PL=8
MOVL C00288 V=800.0 PL=8
MOVL C00289 V=800.0 PL=8
MOVL C00290 V=800.0 PL=0
SPYOF
MOVJ C00291 VJ=25.00 PL=0
SPYON
MOVL C00292 V=800.0 PL=8
MOVL C00293 V=800.0 PL=8
MOVL C00294 V=800.0 PL=8
MOVL C00295 V=800.0 PL=8
MOVL C00296 V=800.0 PL=8
MOVL C00297 V=800.0 PL=8
MOVL C00298 V=800.0 PL=8
MOVL C00299 V=800.0 PL=8
MOVL C00300 V=800.0 PL=8
MOVL C00301 V=800.0 PL=8
MOVL C00302 V=800.0 PL=8
MOVL C00303 V=800.0 PL=8
MOVL C00304 V=800.0 PL=8
MOVL C00305 V=800.0 PL=8
MOVL C00306 V=800.0 PL=8
MOVL C00307 V=800.0 PL=8
MOVL C00308 V=800.0 PL=8
MOVL C00309 V=800.0 PL=8
MOVL C00310 V=800.0 PL=8
MOVL C00311 V=800.0 PL=8
MOVL C00312 V=800.0 PL=8
MOVL C00313 V=800.0 PL=8
MOVL C00314 V=800.0 PL=8
MOVL C00315 V=800.0 PL=8
MOVL C00316 V=800.0 PL=8
MOVL C00317 V=800.0 PL=8
MOVL C00318 V=800.0 PL=8
MOVL C00319 V=800.0 PL=8
MOVL C00320 V=800.0 PL=8
MOVL C00321 V=800.0 PL=8
MOVL C00322 V=800.0 PL=8
MOVL C00323 V=800.0 PL=8
MOVL C00324 V=800.0 PL=8
MOVL C00325 V=800.0 PL=8
MOVL C00326 V=800.0 PL=8
MOVL C00327 V=800.0 PL=8
MOVL C00328 V=800.0 PL=8
MOVL C00329 V=800.0 PL=0
SPYOF
MOVJ C00330 VJ=25.00 PL=0
SPYON
MOVL C00331 V=800.0 PL=8
MOVL C00332 V=800.0 PL=8
MOVL C00333 V=800.0 PL=8
MOVL C00334 V=800.0 PL=8
MOVL C00335 V=800.0 PL=8
MOVL C00336 V=800.0 PL=8
MOVL C00337 V=800.0 PL=8
MOVL C00338 V=800.0 PL=8
MOVL C00339 V=800.0 PL=8
MOVL C00340 V=800.0 PL=8
MOVL C00341 V=800.0 PL=8
MOVL C00342 V=800.0 PL=8
MOVL C00343 V=800.0 PL=8
MOVL C00344 V=800.0 PL=8
MOVL C00345 V=800.0 PL=8
MOVL C00346 V=800.0 PL=8
MOVL C00347 V=800.0 PL=8
MOVL C00348 V=800.0 PL=8
MOVL C00349 V=800.0 PL=8
MOVL C00350 V=800.0 PL=8
MOVL C00351 V=800.0 PL=8
MOVL C00352 V=800.0 PL=8
MOVL C00353 V=800.0 PL=8
MOVL C00354 V=800.0 PL=8
MOVL C00355 V=800.0 PL=8
MOVL C00356 V=800.0 PL=8
MOVL C00357 V=800.0 PL=8
MOVL C00358 V=800.0 PL=8
MOVL C00359 V=800.0 PL=8
MOVL C00360 V=800.0 PL=8
MOVL C00361 V=800.0 PL=8
MOVL C00362 V=800.0 PL=8
MOVL C00363 V=800.0 PL=8
MOVL C00364 V=800.0 PL=8
MOVL C00365 V=800.0 PL=8
MOVL C00366 V=800.0 PL=8
MOVL C00367 V=800.0 PL=8
MOVL C00368 V=800.0 PL=8
MOVL C00369 V=800.0 PL=0
SPYOF
MOVJ C00370 VJ=25.00 PL=0
SPYON
MOVL C00371 V=800.0 PL=8
MOVL C00372 V=800.0 PL=8
MOVL C00373 V=800.0 PL=8
MOVL C00374 V=800.0 PL=8
MOVL C00375 V=800.0 PL=8
MOVL C00376 V=800.0 PL=8
MOVL C00377 V=800.0 PL=8
MOVL C00378 V=800.0 PL=8
MOVL C00379 V=800.0 PL=8
MOVL C00380 V=800.0 PL=8
MOVL C00381 V=800.0 PL=8
MOVL C00382 V=800.0 PL=8
MOVL C00383 V=800.0 PL=8
MOVL C00384 V=800.0 PL=8
MOVL C00385 V=800.0 PL=8
MOVL C00386 V=800.0 PL=8
MOVL C00387 V=800.0 PL=8
MOVL C00388 V=800.0 PL=8
MOVL C00389 V=800.0 PL=8
MOVL C00390 V=800.0 PL=8
MOVL C00391 V=800.0 PL=8
MOVL C00392 V=800.0 PL=8
MOVL C00393 V=800.0 PL=8
MOVL C00394 V=800.0 PL=8
MOVL C00395 V=800.0 PL=8
MOVL C00396 V=800.0 PL=8
MOVL C00397 V=800.0 PL=8
MOVL C00398 V=800.0 PL=8
MOVL C00399 V=800.0 PL=8
MOVL C00400 V=800.0 PL=8
MOVL C00401 V=800.0 PL=8
MOVL C00402 V=800.0 PL=8
MOVL C00403 V=800.0 PL=8
MOVL C00404 V=800.0 PL=8
MOVL C00405 V=800.0 PL=8
MOVL C00406 V=800.0 PL=8
MOVL C00407 V=800.0 PL=8
MOVL C00408 V=800.0 PL=8
MOVL C00409 V=800.0 PL=8
MOVL C00410 V=800.0 PL=8
MOVL C00411 V=800.0 PL=0
SPYOF
MOVJ C00412 VJ=25.00 PL=0
SPYON
MOVL C00413 V=800.0 PL=8
MOVL C00414 V=800.0 PL=8
MOVL C00415 V=800.0 PL=8
MOVL C00416 V=800.0 PL=8
MOVL C00417 V=800.0 PL=8
MOVL C00418 V=800.0 PL=8
MOVL C00419 V=800.0 PL=8
MOVL C00420 V=800.0 PL=8
MOVL C00421 V=800.0 PL=8
MOVL C00422 V=800.0 PL=8
MOVL C00423 V=800.0 PL=8
MOVL C00424 V=800.0 PL=8
MOVL C00425 V=800.0 PL=8
MOVL C00426 V=800.0 PL=8
MOVL C00427 V=800.0 PL=8
MOVL C00428 V=800.0 PL=8
MOVL C00429 V=800.0 PL=8
MOVL C00430 V=800.0 PL=8
MOVL C00431 V=800.0 PL=8
MOVL C00432 V=800.0 PL=8
MOVL C00433 V=800.0 PL=8
MOVL C00434 V=800.0 PL=8
MOVL C00435 V=800.0 PL=8
MOVL C00436 V=800.0 PL=8
MOVL C00437 V=800.0 PL=8
MOVL C00438 V=800.0 PL=8
MOVL C00439 V=800.0 PL=8
MOVL C00440 V=800.0 PL=8
MOVL C00441 V=800.0 PL=8
MOVL C00442 V=800.0 PL=8
MOVL C00443 V=800.0 PL=8
MOVL C00444 V=800.0 PL=8
MOVL C00445 V=800.0 PL=8
MOVL C00446 V=800.0 PL=0
SPYOF
MOVL C00447 V=800.0 PL=8
MOVJ C00448 VJ=25.00 PL=0
SPYON
MOVL C00449 V=800.0 PL=8
MOVL C00450 V=800.0 PL=8
MOVL C00451 V=800.0 PL=8
MOVL C00452 V=800.0 PL=8
MOVL C00453 V=800.0 PL=8
MOVL C00454 V=800.0 PL=8
MOVL C00455 V=800.0 PL=8
MOVL C00456 V=800.0 PL=8
MOVL C00457 V=800.0 PL=8
MOVL C00458 V=800.0 PL=8
MOVL C00459 V=800.0 PL=8
MOVL C00460 V=800.0 PL=0
SPYOF
MOVJ C00461 VJ=25.00 PL=0
SPYON
MOVL C00462 V=800.0 PL=8
MOVL C00463 V=800.0 PL=8
MOVL C00464 V=800.0 PL=8
MOVL C00465 V=800.0 PL=8
MOVL C00466 V=800.0 PL=8
MOVL C00467 V=800.0 PL=0
SPYOF
MOVJ C00468 VJ=25.00 PL=0
SPYON
MOVL C00469 V=800.0 PL=8
MOVL C00470 V=800.0 PL=8
MOVL C00471 V=800.0 PL=8
MOVL C00472 V=800.0 PL=8
MOVL C00473 V=800.0 PL=8
MOVL C00474 V=800.0 PL=0
SPYOF
MOVJ C00475 VJ=25.00 PL=0
'Path End
MOVJ C00476 VJ=25.00 PL=0
END
